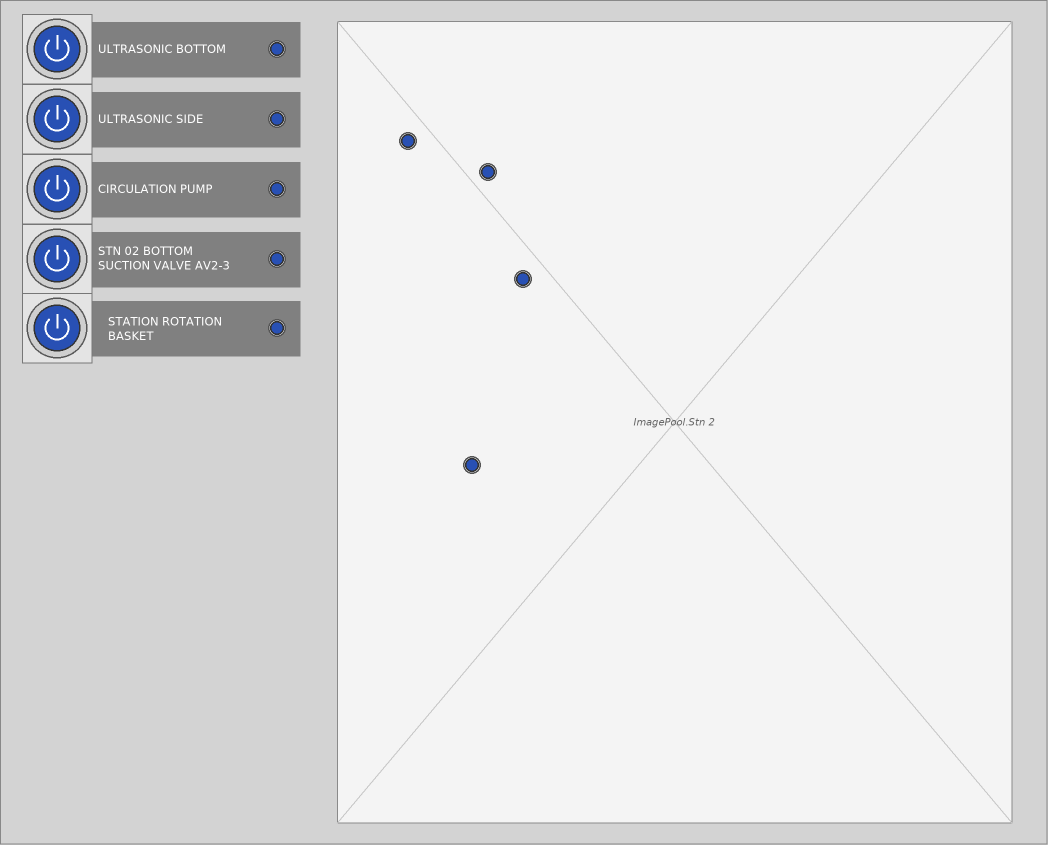
VISUALIZATION Recipe_Station02  // 1048x845
    Rectangle (0,0 1048x845)
    Image (337,21 675x802), image: ImagePool.Stn 2
    RoundedRectangle (61,22 239x55)
    Label (95,41 163x16), "ULTRASONIC BOTTOM"
    Lamp1 (267,39 20x20), variable: DSScrMapSSUR.DsSubRecipeMemory.bOut3EnProTankBottomUltrasonicA, style: Lamp-Lamp1-Blue
    PowerSwitch (22,14 70x70), variable: DSScrMapSSUR.DsSubRecipeMemory.bOut3EnProTankBottomUltrasonicA, behaviour: TOGGLE, style: Switch-PowerSwitch-Blue
    RoundedRectangle (69,162 231x55)
    Label (95,181 151x16), "CIRCULATION PUMP"
    Lamp1 (267,179 20x20), variable: DSScrMapSSUR.DsSubRecipeMemory.bOut1EnProTankPump, style: Lamp-Lamp1-Blue
    PowerSwitch (22,154 70x70), variable: DSScrMapSSUR.DsSubRecipeMemory.bOut1EnProTankPump, behaviour: TOGGLE, style: Switch-PowerSwitch-Blue
    RoundedRectangle (69,232 231x55)
    Label (95,244 151x29), "STN 02 BOTTOM SUCTION VALVE AV2-3"
    Lamp1 (267,249 20x20), variable: DSScrMapSSUR.DsSubRecipeMemory.bOut3ActValve3, style: Lamp-Lamp1-Blue
    PowerSwitch (22,224 70x70), variable: DSScrMapSSUR.DsSubRecipeMemory.bOut3ActValve3, behaviour: TOGGLE, style: Switch-PowerSwitch-Blue
    RoundedRectangle (61,92 239x55)
    Label (95,111 163x16), "ULTRASONIC SIDE"
    Lamp1 (267,109 20x20), variable: DSScrMapSSUR.DsSubRecipeMemory.bOut6EnProTankSideUltrasonicA, style: Lamp-Lamp1-Blue
    PowerSwitch (22,84 70x70), variable: DSScrMapSSUR.DsSubRecipeMemory.bOut6EnProTankSideUltrasonicA, behaviour: TOGGLE, style: Switch-PowerSwitch-Blue
    Lamp1 (478,162 20x20), variable: DSScrMapSSUR.DsSubRecipeMemory.bOut3EnProTankBottomUltrasonicA, style: Lamp-Lamp1-Blue
    Lamp1 (462,455 20x20), variable: DSScrMapSSUR.DsSubRecipeMemory.bOut1EnProTankPump, style: Lamp-Lamp1-Blue
    Lamp1 (513,269 20x20), variable: DSScrMapSSUR.DsSubRecipeMemory.bOut3ActValve3, style: Lamp-Lamp1-Blue
    Lamp1 (398,131 20x20), variable: DSScrMapSSUR.DsSubRecipeMemory.bOut6EnProTankSideUltrasonicA, style: Lamp-Lamp1-Blue
    RoundedRectangle (69,301 231x55)
    Lamp1 (267,318 20x20), variable: DSScrMapSSUR.DsSubRecipeMemory.bOut14EnInstrument3, style: Lamp-Lamp1-Blue
    PowerSwitch (22,293 70x70), variable: DSScrMapSSUR.DsSubRecipeMemory.bOut14EnInstrument3, behaviour: TOGGLE, style: Switch-PowerSwitch-Blue
    Label (105,312 151x34), "STATION ROTATION BASKET"
END_VISUALIZATION

(* stored: Version 1.1.0.1, ProductVersion 3.1.4024.12
   Visu Recipe_Station02: Id {958168f4-5fd1-4dab-906a-83857df40a79} *)
